// TIA Portal V18 export
TYPE "User_data_type_2"
// stored: IsFailsafeCompliant false
   STRUCT
      on : Bool;
      off : Bool;
      lamp : Bool;
   END_STRUCT;
END_TYPE
